FUNCTION_BLOCK fbLIT
VAR_INPUT
	In : REAL;
END_VAR
VAR_OUTPUT
	Level : REAL;
	WarningLow : BOOL;
	AlarmLow : BOOL;
	WarningHigh : BOOL;
	AlarmHigh : BOOL;
END_VAR
VAR
	LLLimit : REAL := 10;
	LLimit : REAL := 20;
	HLimit : REAL := 80;
	HHLimit : REAL := 90;
	AlarmDelay : DINT := 10; // Alarm Delay in secondss
	HHDelayTON : TON;
	HDelayTON : TON;
	LDelayTON : TON;
	LLDelayTON : TON;
	tAlarmDelay: TIME;
END_VAR

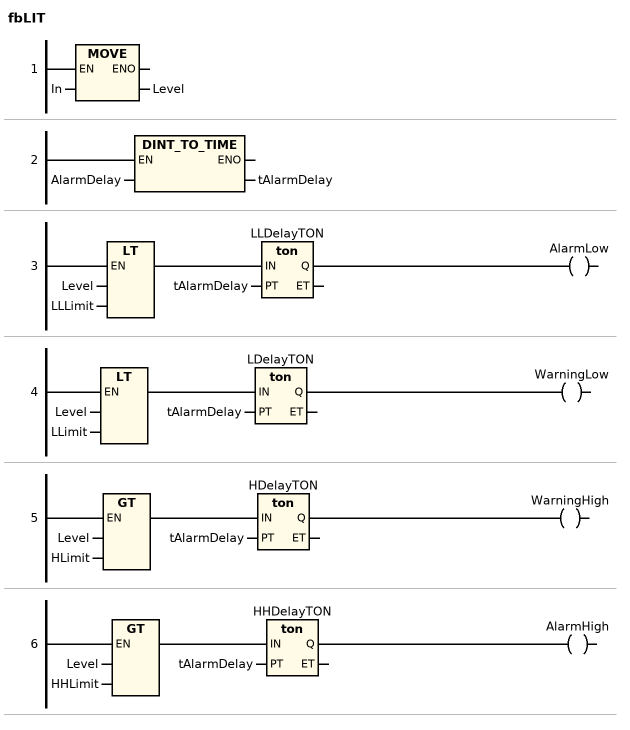
// NETWORK 1
Level := In;

// NETWORK 2
tAlarmDelay := DINT_TO_TIME(AlarmDelay);

// NETWORK 3
LLDelayTON(IN := Level < LLLimit, PT := tAlarmDelay); // ton
AlarmLow := LLDelayTON.Q;

// NETWORK 4
LDelayTON(IN := Level < LLimit, PT := tAlarmDelay); // ton
WarningLow := LDelayTON.Q;

// NETWORK 5
HDelayTON(IN := Level > HLimit, PT := tAlarmDelay); // ton
WarningHigh := HDelayTON.Q;

// NETWORK 6
HHDelayTON(IN := Level > HHLimit, PT := tAlarmDelay); // ton
AlarmHigh := HHDelayTON.Q;

END_FUNCTION_BLOCK

(* stored: Version 1.1.0.1, ProductVersion 3.1.4022.17
   POU fbLIT: Id {e650c7d0-c4e7-4e05-b638-70a2c8c649f3}, SpecialFunc None *)
